FUNCTION_BLOCK FB_Motor
VAR_INPUT
	bLiga, bDesliga, bReset:BOOL;
	rTemp:REAL;
END_VAR
VAR_OUTPUT
	bLigaMotor, bError:BOOL;
END_VAR
VAR
END_VAR

IF rTemp >=100 THEN
	bError:=TRUE;
END_IF
IF bLiga AND NOT bDesliga AND NOT bError AND rTemp<80 THEN
	bLigaMotor:=TRUE;
ELSIF bDesliga OR bError THEN
	bLigaMotor:=FALSE;
END_IF

IF bReset AND rTemp < 80 THEN
	bError:=FALSE;
END_IF

END_FUNCTION_BLOCK

(* stored: Version 1.1.0.1, ProductVersion 3.1.4024.11
   POU FB_Motor: Id {794e1372-b388-4a05-ba78-6561b776a7a6}, SpecialFunc None *)
